# B&R Automation Studio project POM-RS2
Automation Studio 4.5.2.102

## Configuration Config1

### Task classes (Cpu.sw)
```
Cyclic#1 (cycle 2000 us):
  Program <- Program.prg
NcDataObjects: acp10etxen <- acp10etxen.dob
Libraries: Acp10man, Acp10par, NcGlobal, Acp10sdc, AsBrStr, DriveLib
```

### Hardware
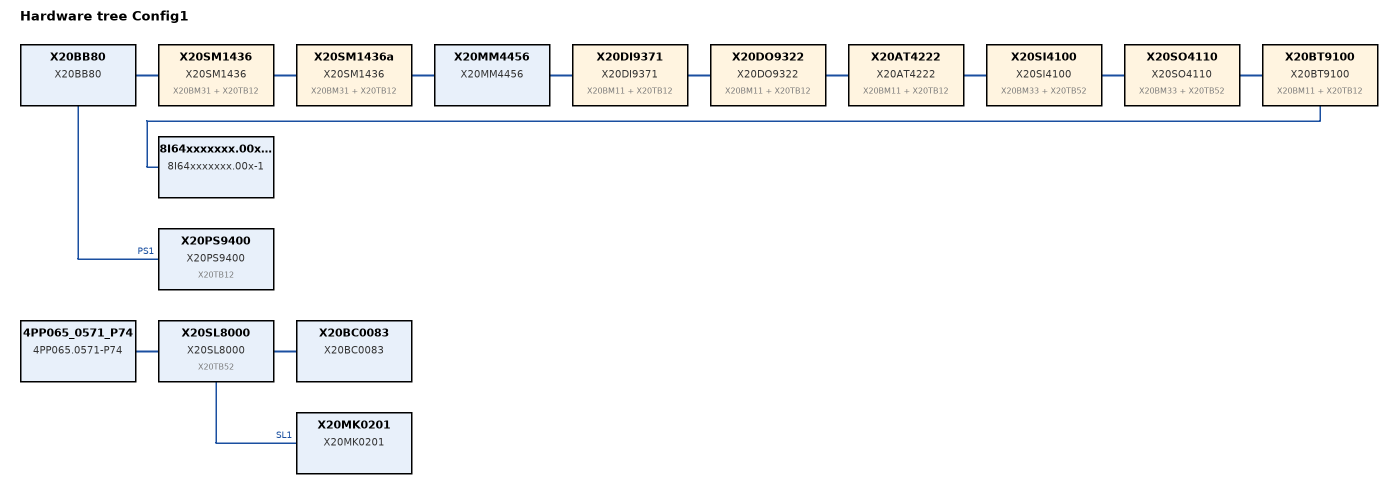
```
4PP065_0571_P74 : 4PP065.0571-P74 v1.1.2.0
  Connector IF5:
    ActivateDevice = 1
    Mode = Manual
    InternetAddress = 10.0.1.10
    SubnetMask = 255.255.255.0
  ConfigurationID = labBR
  TimerDeviceType = EPLX2X
  TimerDevice = 4PP065_0571_P74.IF4
  TaskClassIdleTime = 2000
  Cyclic1Duration = 2000
  Cyclic1Output = 1
8I64xxxxxxx.00x-1 : 8I64xxxxxxx.00x-1 v1.3.9.1  [X2X1 -> X20BT9100.X2X1 [Cable Type=X2XCable, Length=10, Version=1.0.0.2]]
  FunctionModel = Standard
  packedETAD = packed
  packedETI = packed
  packedCMDD = packed
  packedCMI = packed
  UNS = 220
  NCR = 10
  NSP = 890
  COS = 64
  RSC = 33000
X20AT4222 : X20AT4222 v1.2.3.0  [SS1 -> X20TB12e.SS; SL -> X20BM11b.SL1]
X20BB80 : X20BB80 v1.0.2.0
X20BC0083 : X20BC0083 v2.7.0.0  [PLK1 -> X20SL8000.PLK2 [Cable Type=PowerlinkCable, Length=10, Version=1.0.0.2]; SL -> X20BB80.SL1]
X20BM11 : X20BM11 v1.0.0.1  [X2X1 -> X20MM4456.X2X2]
X20BM11a : X20BM11 v1.0.0.1  [X2X1 -> X20BM11.X2X2]
X20BM11b : X20BM11 v1.0.0.1  [X2X1 -> X20BM11a.X2X2]
X20BM11c : X20BM11 v1.0.0.1  [X2X1 -> X20BM33a.X2X2]
X20BM31 : X20BM31 v1.0.0.1  [X2X1 -> X20BB80.IF1]
X20BM31a : X20BM31 v1.0.0.1  [X2X1 -> X20BM31.X2X2]
X20BM33 : X20BM33 v1.0.0.4  [X2X1 -> X20BM11b.X2X2]
X20BM33a : X20BM33 v1.0.0.4  [X2X1 -> X20BM33.X2X2]
X20BT9100 : X20BT9100 v1.0.3.0  [SS1 -> X20TB12f.SS; SL -> X20BM11c.SL1]
X20DI9371 : X20DI9371 v1.0.2.0  [SS1 -> X20TB12c.SS; SL -> X20BM11.SL1]
X20DO9322 : X20DO9322 v1.0.3.0  [SS1 -> X20TB12d.SS; SL -> X20BM11a.SL1]
X20MK0201 : X20MK0201 v1.0.0.0  [SL -> X20SL8000.SL1]
X20MM4456 : X20MM4456 v1.1.5.0  [X2X1 -> X20BM31a.X2X2]
X20PS9400 : X20PS9400 v1.0.2.4  [SS1 -> X20TB12.SS; PS -> X20BB80.PS1]
X20SI4100 : X20SI4100 v1.10.1.1  [SS1 -> X20TB52a.SS; SL -> X20BM33.SL1]
X20SL8000 : X20SL8000 v1.6.5.1  [PLK1 -> 4PP065_0571_P74.IF4 [Cable Type=PowerlinkCable, Length=10, Version=1.0.0.2]; PLK2 -> X20BC0083.PLK1 [Cable Type=PowerlinkCable, Length=10, Version=1.0.0.2]; SS1 -> X20TB52.SS]
  SafeProject = SafeLOGIC-1
X20SM1436 : X20SM1436 v1.4.2.1  [SS1 -> X20TB12a.SS; SL -> X20BM31.SL1]
X20SM1436a : X20SM1436 v1.4.2.1  [SS1 -> X20TB12b.SS; SL -> X20BM31a.SL1]
X20SO4110 : X20SO4110 v1.10.1.1  [SS1 -> X20TB52b.SS; SL -> X20BM33a.SL1]
  SafeModuleID = 3
X20TB12 : X20TB12 v1.0.0.0
X20TB12a : X20TB12 v1.0.0.0
X20TB12b : X20TB12 v1.0.0.0
X20TB12c : X20TB12 v1.0.0.0
X20TB12d : X20TB12 v1.0.0.0
X20TB12e : X20TB12 v1.0.0.0
X20TB12f : X20TB12 v1.0.0.0
X20TB52 : X20TB52 v1.0.0.1
X20TB52a : X20TB52 v1.0.0.1
X20TB52b : X20TB52 v1.0.0.1
```

### IoMap.iom - 4PP065_0571_P74/IoMap.iom
```iecst
VAR_CONFIG
	::Program:driveSM.state AT %IW."8I64xxxxxxx.00x-1".ETAD_Input;
	::Program:driveSM.command AT %QW."8I64xxxxxxx.00x-1".CMDD_Output;
	::Program:driveSM.speed AT %QW."8I64xxxxxxx.00x-1".LFRD_Output;
	::Program:doorSM.direction AT %IX."X20DI9371".DigitalInput01;
	::Program:doorSM.sw[3] AT %IX."X20DI9371".DigitalInput02;
	::Program:doorSM.sw[2] AT %IX."X20DI9371".DigitalInput03;
	::Program:doorSM.sw[1] AT %IX."X20DI9371".DigitalInput04;
	::Program:doorSM.sw[0] AT %IX."X20DI9371".DigitalInput05;
	::Program:ledSM.led[3] AT %QX."X20DO9322".DigitalOutput02;
	::Program:ledSM.led[2] AT %QX."X20DO9322".DigitalOutput03;
	::Program:ledSM.led[1] AT %QX."X20DO9322".DigitalOutput04;
	::Program:ledSM.led[0] AT %QX."X20DO9322".DigitalOutput05;
	::Program:driveSM.speedFeedback AT %IW."8I64xxxxxxx.00x-1".RFRD_Input;
END_VAR
```

## Logical view

Binary libraries used (declarations not repeated): operator, runtime, astime, AsIecCon, Acp10man, Acp10par, NcGlobal, Acp10sdc, AsBrStr

### Global.var - Global variables
```iecst
VAR
	count : USINT;
END_VAR
```

### Package Logical/Libraries - Global libraries

### Library Logical/Libraries/DriveLib (ANSIC)

#### Types.typ - Exported data types
```iecst
TYPE
	DoorStates :
		(
		ST_INIT,
		ST_UNKNOWN,
		ST_OPEN,
		ST_CLOSE,
		ST_ACC_POS,
		ST_ACC_NEG,
		ST_POS,
		ST_NEG,
		ST_DEC_POS,
		ST_DEC_NEG
		);
	DriveStates :
		(
		ST_DISABLED := 64,
		ST_SWITCHED_ON := 35,
		ST_READY := 33
		);
	DriveCommands :
		(
		CMD_ENABLE := 15,
		CMD_SWITCH_ON := 7,
		CMD_SHUTDOWN := 6
		);
END_TYPE
```

#### Constants.var - Exported constants
```iecst
VAR CONSTANT
	maxSpeed : INT := 890;
	minSpeed : INT := 89;
	maxFreq : USINT := 10;
	cycleTime : USINT := 2;
END_VAR
```

#### DriveLib.fun - Exported functions and function blocks
```iecst
FUNCTION_BLOCK DoorStateMachine
	VAR_INPUT
		state : DoorStates;
		direction : BOOL;
		sw : ARRAY[0..3] OF BOOL;
	END_VAR
	VAR_OUTPUT
		speed : INT;
	END_VAR
	VAR
		sw_prev : ARRAY[0..3] OF BOOL;
		sw_pressed : ARRAY[0..3] OF BOOL;
	END_VAR
END_FUNCTION_BLOCK

FUNCTION_BLOCK DriveStateMachine
	VAR_INPUT
		state : UINT;
		enable : BOOL;
		speed : INT;
	END_VAR
	VAR_OUTPUT
		command : UINT;
		speedFeedback : INT;
	END_VAR
END_FUNCTION_BLOCK

FUNCTION_BLOCK LedStateMachine
	VAR_INPUT
		state : DoorStates;
		speed : INT;
	END_VAR
	VAR_OUTPUT
		led : ARRAY[0..3] OF BOOL;
	END_VAR
	VAR
		count : UINT;
	END_VAR
END_FUNCTION_BLOCK

{REDUND_ERROR} FUNCTION SpeedToFreq : USINT (*TODO: Add your comment here*) (*$GROUP=User,$CAT=User,$GROUPICON=User.png,$CATICON=User.png*)
	VAR_INPUT
		speed : INT;
	END_VAR
END_FUNCTION
```

#### DoorStateMachine.c
```c
#include <bur/plctypes.h>
#ifdef __cplusplus
	extern "C"
	{
#endif
#include "DriveLib.h"
#ifdef __cplusplus
	};
#endif
/* TODO: Add your comment here */
void DoorStateMachine(struct DoorStateMachine* inst)
{
	switch (inst->state)
	{
		case ST_INIT:
			inst->state = ST_UNKNOWN;
			break;
		case ST_UNKNOWN:
			if (inst->direction == 1)
				inst->speed = maxSpeed / 5;
			else
				inst->speed = -maxSpeed / 5;

			if (inst->direction == 0 && inst->sw[0] != inst->sw_prev[0])
			{
				inst->state = ST_OPEN;
				inst->speed = 0;
			}
			else if (inst->direction == 1 && inst->sw[3] != inst->sw_prev[3])
			{
				inst->state = ST_CLOSE;
				inst->speed = 0;
			}
			break;
		case ST_OPEN:
			if (inst->direction == 1)
			{
				inst->state = ST_ACC_POS;
				inst->speed = minSpeed;
			}
			break;
		case ST_ACC_POS:
			if (inst->sw[1] != inst->sw_prev[1])
			{
				inst->state = ST_POS;
				inst->speed = maxSpeed / 2;
			}
			else if (inst->direction == 0)
			{
				inst->state = ST_DEC_NEG;
				inst->speed = -minSpeed;
			}
			break;
		case ST_POS:
			if (inst->sw[2] != inst->sw_prev[2])
			{
				inst->state = ST_DEC_POS;
				inst->speed = minSpeed;
			}
			else if (inst->direction == 0)
			{
				inst->state = ST_NEG;
				inst->speed = -maxSpeed / 2;
			}
			break;
		case ST_DEC_POS:
			if (inst->sw[3] != inst->sw_prev[3])
			{
				inst->state = ST_CLOSE;
				inst->speed = 0;
			}
			else if (inst->direction == 0)
			{
				inst->state = ST_ACC_NEG;
				inst->speed = -minSpeed;
			}
			break;
		case ST_CLOSE:
			if (inst->direction == 0)
			{
				inst->state = ST_ACC_NEG;
				inst->speed = -minSpeed;
			}
			break;
		case ST_ACC_NEG:
			if (inst->sw[2] != inst->sw_prev[2])
			{
				inst->state = ST_NEG;
				inst->speed = -maxSpeed / 2;
			}
			else if (inst->direction == 1)
			{
				inst->state = ST_DEC_POS;
				inst->speed = minSpeed;
			}
			break;
		case ST_NEG:
			if (inst->sw[1] != inst->sw_prev[1])
			{
				inst->state = ST_DEC_NEG;
				inst->speed = -minSpeed;
			}
			else if (inst->direction == 1)
			{
				inst->state = ST_POS;
				inst->speed = maxSpeed / 2;
			}
			break;
		case ST_DEC_NEG:
			if (inst->sw[0] != inst->sw_prev[0])
			{
				inst->state = ST_OPEN;
				inst->speed = 0;
			}
			else if (inst->direction == 1)
			{
				inst->state = ST_ACC_POS;
				inst->speed = minSpeed;
			}
			break;
	}

	//memorizing states' switch for buttons
	int i;
	for (i = 0; i < 4; i++)
	{
		inst->sw_pressed[i] = (inst->sw[i] != inst->sw_prev[i]);
		inst->sw_prev[i] = inst->sw[i];
	}
}
```

#### DriveStateMachine.c
```c
#include <bur/plctypes.h>
#ifdef __cplusplus
	extern "C"
	{
#endif
#include "DriveLib.h"
#ifdef __cplusplus
	};
#endif
/* TODO: Add your comment here */
void DriveStateMachine(struct DriveStateMachine* inst)
{
	if (!inst->enable)
	{
		inst->command = CMD_SHUTDOWN;
	}
	else
	{
		switch (inst->state & 0x6F)
		{
			case ST_DISABLED:
				inst->command = CMD_SHUTDOWN;
				break;
			case ST_READY:
				inst->command = CMD_ENABLE;
				break;
			case ST_SWITCHED_ON:
				inst->command = CMD_SWITCH_ON;
				break;
		}
	}
}
```

#### LedStateMachine.c
```c
#include <bur/plctypes.h>
#ifdef __cplusplus
	extern "C"
	{
#endif
#include "DriveLib.h"
#ifdef __cplusplus
	};
#endif
/* TODO: Add your comment here */
void LedStateMachine(struct LedStateMachine* inst)
{
	inst->count++;
	int i;
	switch (inst->state)
	{
		case ST_INIT:
			for (i = 0; i < 4; i++)
				inst->led[i] = 0;
			break;
		case ST_UNKNOWN:
			if (inst->count % (500 / cycleTime) == 0)
			{
				for (i = 0; i < 4; i++)
					inst->led[i] = !inst->led[i];
			}
			break;
		case ST_OPEN:
			for (i = 0; i < 4; i++)
				inst->led[i] = 0;
			break;
		case ST_ACC_POS:
			inst->led[3] = 0;
			inst->led[2] = 0;
			if (inst->count % (500 / (cycleTime * SpeedToFreq(inst->speed))) == 0)
				inst->led[1] = !inst->led[1];
			inst->led[0] = 1;
			break;
		case ST_POS:
			inst->led[3] = 0;
			if (inst->count % (500 / (cycleTime * SpeedToFreq(inst->speed))) == 0)
				inst->led[2] = !inst->led[2];
			inst->led[1] = 1;
			inst->led[0] = 1;
			break;
		case ST_DEC_POS:
			if (inst->count % (500 / (cycleTime * SpeedToFreq(inst->speed))) == 0)
				inst->led[3] = !inst->led[3];
			inst->led[2] = 1;
			inst->led[1] = 1;
			inst->led[0] = 1;
			break;
		case ST_CLOSE:
			for (i = 0; i < 4; i++)
				inst->led[i] = 1;
			break;
		case ST_ACC_NEG:
			inst->led[3] = 0;
			if (inst->count % (500 / (cycleTime * SpeedToFreq(inst->speed))) == 0)
				inst->led[2] = !inst->led[2];
			inst->led[1] = 1;
			inst->led[0] = 1;
			break;
		case ST_NEG:
			inst->led[3] = 0;
			inst->led[2] = 0;
			if (inst->count % (500 / (cycleTime * SpeedToFreq(inst->speed))) == 0)
				inst->led[1] = !inst->led[1];
			inst->led[0] = 1;
			break;
		case ST_DEC_NEG:
			inst->led[3] = 0;
			inst->led[2] = 0;
			inst->led[1] = 0;
			if (inst->count % (500 / (cycleTime * SpeedToFreq(inst->speed))) == 0)
				inst->led[0] = !inst->led[0];
			break;
	}
}
```

#### SpeedToFreq.c
```c
#include <bur/plctypes.h>
#ifdef __cplusplus
	extern "C"
	{
#endif
	#include "DriveLib.h"
#ifdef __cplusplus
	};
#endif
/* TODO: Add your comment here */
unsigned char SpeedToFreq(signed short speed)
{
	return maxFreq * (speed > 0 ? speed : -speed) / maxSpeed;
}
```

### Program Logical/Program (ANSIC)

#### Variables.var
```iecst
VAR
	driveSM : DriveStateMachine;
	doorSM : DoorStateMachine;
	ledSM : LedStateMachine;
END_VAR
```

#### Main.c
```c
#include <bur/plctypes.h>

#ifdef _DEFAULT_INCLUDES
	#include <AsDefault.h>
#endif

void _INIT ProgramInit(void)
{
	doorSM.state = ST_INIT;

	int i;
	for (i = 0; i < 4; i++)
		doorSM.sw_prev[i] = doorSM.sw[i];
}

void _CYCLIC ProgramCyclic(void)
{
	doorSM.direction = !doorSM.direction;

	DoorStateMachine(&doorSM);

	driveSM.enable = 1;
	driveSM.speed = doorSM.speed;
	DriveStateMachine(&driveSM);

	ledSM.state = doorSM.state;
	ledSM.speed = doorSM.speed;
	LedStateMachine(&ledSM);
}

void _EXIT ProgramExit(void)
{

}
```

Listed in the project but not available here: Logical/Global.typ, Logical/acp10etxen
